FUNCTION F_WeightCalc : real
VAR_INPUT
	dia			: REAL;
	height 		: REAL;
END_VAR
VAR
END_VAR

F_WeightCalc := dia*pi*height;

END_FUNCTION

(* stored: Version 1.1.0.1, ProductVersion 3.1.4024.12
   POU F_WeightCalc: Id {2b206187-600e-4336-b998-08e78e06b406}, SpecialFunc None *)
